// TIA Portal V17 export
// export: Created 2023-09-10T16:27:53.2673646Z, ExportSetting WithDefaults, DisplayName Totally Integrated Automation Portal, DisplayVersion V17, DisplayName TIA Portal Openness, DisplayVersion V17, DisplayName TIA Portal Version Control Interface, DisplayVersion V17, DisplayName STEP 7 Professional, DisplayVersion V17, DisplayName STEP 7 Safety, DisplayVersion V17, DisplayName WinCC Advanced, DisplayVersion V17
DATA_BLOCK "speedDirectionCalculation_DB"   // DB9
VERSION : 0.1
// stored: AutoNumber true, DBAccessibleFromOPCUA true, InstanceOfName speedDirectionCalculation, InstanceOfType FB
"speedDirectionCalculation"
   // VAR_INPUT
   //    setpointSource : Bool;
   //    setpoint : Int;
   //    serwisSetpoint : DInt;
   //    machineConst : Real;
   //    machinePosition : DInt;
   //    machineSpeed : Int;
   //    manualSpeed : Int;
   //    baseSpeed : Int;
   //    homingSeq : Int;
   //    goToSetpoint : Bool;
   //    jog : Bool;
   // END_VAR
   // VAR_OUTPUT
   //    stepperMotorDirection : Bool;
   //    inRequestPosition : Bool;
   //    speedForStepperMotor : Real;
   //    reqPositionValue : DInt;
   // END_VAR
   // VAR
   //    reqPosition : Real;
   // END_VAR
BEGIN
END_DATA_BLOCK
